FUNCTION_BLOCK FB_Example
VAR
    IFace : BOOL;
    bTHENx : BOOL;
END_VAR
BEGIN
IFace := TRUE;
bTHENx := FALSE;
END_FUNCTION_BLOCK
